FUNCTION_BLOCK LED_ON (* Service Interface Function Block Type *)
  (* Standard: 61499-2 *)
  (* Version 1.0, 2025-05-16, dmitry *)
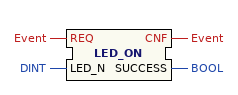
  EVENT_INPUT
    REQ; (* Service Request *)
  END_EVENT
  EVENT_OUTPUT
    CNF; (* Confirmation of Requested Service *)
  END_EVENT
  VAR_INPUT
    LED_N : DINT; (* Led number *)
  END_VAR
  VAR_OUTPUT
    SUCCESS : BOOL;
  END_VAR
  (* Service APPLICATION/RESOURCE: Service Interface Function Block Type *)
END_FUNCTION_BLOCK
